// TIA Portal V18 export
// export: Created 2025-12-01T12:38:32.3552566Z, ExportSetting None, DisplayName Totally Integrated Automation Portal, DisplayVersion V18 Update 5, DisplayName TIA Portal Openness, DisplayVersion V18 Update 5, DisplayName TIA Portal Teamcenter Gateway, DisplayVersion V18, DisplayName TIA Portal Version Control Interface, DisplayVersion V18, DisplayName STEP 7 Professional, DisplayVersion V18 Update 5, DisplayName STEP 7 Safety, DisplayVersion V18, DisplayName WinCC Professional, DisplayVersion V18 Update 5
DATA_BLOCK "ST10_PMCountCycleTime"   // DB1061
{ S7_Optimized_Access := 'FALSE' }
// stored: AutoNumber false
   VAR
      PM : Array[1..30] of "RCS_CountCycleTime_V1";
      PM_Num : Int;
   END_VAR
BEGIN
END_DATA_BLOCK
